FUNCTION_BLOCK FB_AllocateAreaWithXPlanar EXTENDS FB_ModeBase_V1
VAR_INPUT
	
END_VAR
VAR_OUTPUT
END_VAR
VAR
	UnitInput :REFERENCE TO ST_AllocateInput;
	UnitOutput: REFERENCE TO ST_AllocateOutput;
END_VAR

{attribute 'object_name' := 'M_Aborted'}
METHOD M_Aborted 
VAR_INPUT
END_VAR
END_METHOD

{attribute 'object_name' := 'M_Aborting'}
METHOD M_Aborting
VAR_INPUT
END_VAR
END_METHOD

{attribute 'object_name' := 'M_Clearing'}
METHOD M_Clearing
VAR_INPUT
END_VAR
END_METHOD

{attribute 'object_name' := 'M_Complete'}
METHOD M_Complete
VAR_INPUT
END_VAR
END_METHOD

{attribute 'object_name' := 'M_Completing'}
METHOD M_Completing
VAR_INPUT
END_VAR
END_METHOD

{attribute 'object_name' := 'M_Execute'}
METHOD M_Execute
VAR_INPUT
END_VAR
M_StateComplete();
END_METHOD

{attribute 'object_name' := 'M_Held'}
METHOD M_Held
VAR_INPUT
END_VAR
END_METHOD

{attribute 'object_name' := 'M_Holding'}
METHOD M_Holding
VAR_INPUT
END_VAR
END_METHOD

{attribute 'object_name' := 'M_Idle'}
METHOD M_Idle
VAR_INPUT
END_VAR
END_METHOD

METHOD M_IOMapping
VAR_INPUT
END_VAR
//UnitInput := GVL_in
END_METHOD

{attribute 'object_name' := 'M_Resetting'}
METHOD M_Resetting
VAR_INPUT
END_VAR
END_METHOD

{attribute 'object_name' := 'M_Starting'}
METHOD M_Starting
VAR_INPUT
END_VAR
VAR
	uiStartingStep : DINT;
END_VAR
CASE eMode OF
    E_Mode.Auto:
        CASE uiStartingStep OF
            0: //
            1: //
            2: //
            3: //
            9900:
                M_StateComplete();
        END_CASE
END_CASE
END_METHOD

{attribute 'object_name' := 'M_Stopped'}
METHOD M_Stopped
VAR_INPUT
END_VAR
END_METHOD

{attribute 'object_name' := 'M_Stopping'}
METHOD M_Stopping
VAR_INPUT
END_VAR
END_METHOD

{attribute 'object_name' := 'M_Suspended'}
METHOD M_Suspended
VAR_INPUT
END_VAR
END_METHOD

{attribute 'object_name' := 'M_Suspending'}
METHOD M_Suspending
VAR_INPUT
END_VAR
END_METHOD

{attribute 'object_name' := 'M_Undefined'}
METHOD M_Undefined
VAR_INPUT
END_VAR
END_METHOD

{attribute 'object_name' := 'M_Unholding'}
METHOD M_Unholding
VAR_INPUT
END_VAR
END_METHOD

{attribute 'object_name' := 'M_Unsuspending'}
METHOD M_Unsuspending
VAR_INPUT
END_VAR
END_METHOD

END_FUNCTION_BLOCK

(* stored: Version 1.1.0.1, ProductVersion 3.1.4024.13
   POU FB_AllocateAreaWithXPlanar: Id {99e40695-2fb7-4e99-82ba-c692917c1e16}, SpecialFunc None
   Folder States: Id {adc90e19-bdd2-433c-a576-5132af21cb9e}
   Method M_Aborted: Id {fd178b4e-faae-4ffb-b6bf-939a26de60f2}
   Method M_Aborting: Id {5a02bda1-ac00-4e99-b01c-64ce1262b592}
   Method M_Clearing: Id {c293a841-89a8-4b94-943c-4546b240f3d7}
   Method M_Complete: Id {d932e01d-f79c-4f08-b634-3824b20a6747}
   Method M_Completing: Id {863a44c2-4519-4469-9fe6-c898cef3e302}
   Method M_Execute: Id {445403a2-2f82-4e1a-abea-5df627798d00}
   Method M_Held: Id {88a3f3b0-487b-49d9-b45f-5210c2b694c4}
   Method M_Holding: Id {1c225b28-e445-4a5b-a3ed-ef6831271c97}
   Method M_Idle: Id {5e3c8673-f6e7-482a-8cb9-ece8e323d52c}
   Method M_IOMapping: Id {8c57a45e-2c43-40c5-85bd-c6183955c7e1}
   Method M_Resetting: Id {4d2600c5-7991-4f73-b370-fdd99f5a1042}
   Method M_Starting: Id {04cc518f-8d40-4b06-a44b-b6b73dca765a}
   Method M_Stopped: Id {20bdf14d-d302-452a-a823-b9e7ccca1d11}
   Method M_Stopping: Id {5c479a1d-e94e-44b8-8e59-1da38c86cfaa}
   Method M_Suspended: Id {fecd3ca6-4895-4309-96a3-184929305969}
   Method M_Suspending: Id {af40843d-ce31-4796-b692-cd030fd68611}
   Method M_Undefined: Id {fa0bf4eb-85c3-4394-b849-1686589ad908}
   Method M_Unholding: Id {b3839f71-146b-490c-95c2-ac491920449e}
   Method M_Unsuspending: Id {36f55923-0380-4bf3-9815-97aaf22e7e60} *)
